(* Logix 5000 project; controller cal1615 1756-L62 rev 20.19; software revision 20.05; part 34 of 82 *)
(* tags used below, declared in another part *)
   aaa_prs : REAL;
   FAULT : BOOL;   // Fault AFI
   HMI : BOOL;   // AFI HMI
   p01r09_pb_global_reset : BOOL;   // System Modes PB: Global Fault Reset
   p19_ai_prs : REAL;   // Advanced Cooling Analog Input Pressure [PSI]
   p19_ai_tc01 : REAL;   // Advanced Cooling Analog Input Control Temperature 1
   p19_ao_cv : REAL;   // Advanced Cooling Analog Output Control Valve
   p19_di_tc01_bo : BOOL;   // Advanced Cooling Digital Input Control Thermocouple 1 Failure
   p19_di_tc02_bo : BOOL;   // Advanced Cooling Digital Input Control Thermocouple 2 Failure
   p19_dint_to_hmi : DINT[16];
   p19_do_pump : BOOL;   // Advanced Cooling Digital Output Enable Pump
   p19_flow_input_max : REAL;
   p19_flow_input_min : REAL;
   p19_flow_output_max : REAL;
   p19_flow_output_min : REAL;
   p19_param_pid2_ff : REAL;
   p19_param_pid2_kd : REAL;
   p19_param_pid2_ki : REAL;
   p19_param_pid2_kp : REAL;
   p19_param_tc01_dev : REAL;
   p19_param_tc01z : REAL;   // Advanced Cooling Parameter Control Temperature 1 Zero Offset
   p19_param_tc02z : REAL;   // Advanced Cooling Parameter Control Temperature 2 Zero Offset
   p19_param_zone_pressure : REAL;   // Advanced Cooling Parameter Minimum Pressusre
   p19_prs_input_max1 : REAL;
   p19_prs_input_min1 : REAL;
   p19_prs_output_max1 : REAL;
   p19_prs_output_min1 : REAL;
   p19_real_to_hmi : REAL[80];   // Advanced Cooling Real to HMI
   p19r01 : routine;   // Advanced Cooling Main
   p19r03_flow_scp : SYS_SCP;   // Advanced Cooling Output Roll Cooling Flow Control
   p19r03_prs_scp : SYS_SCP;   // Advanced Cooling Output Cooling Pressure Control Valve Output
   p19r04 : routine;   // Advanced Cooling Output
   p19r04_timer_fault : TIMER[4];   // Advanced Cooling Output Fault Delay
   p19r04_timer_warning : TIMER[4];   // Advanced Cooling Output Warning Delay
   p19r05 : routine;   // Advanced Cooling Dint to HMI
   p19r05_timer_fault : TIMER[4];   // Advanced Cooing Dint to HMI
   p19r05_timer_warning : TIMER[4];   // Advanced Cooling Dint to HMI Warning Delay
   p19r06 : routine;   // Advanced Cooling Real to HMI
   p19r06_timer_fault : TIMER[4];   // Advanced Cooling Real to HMI Fault Delay
   p19r06_timer_warning : TIMER[4];   // Advanced Cooling Real to HMI Warning Delay
   p19r30_cv_man_sp : REAL;   // Advanced Cooling Manual Control Valve Setpoint
   p19r30_pid_temp : PID;   // Advanced Cooling Temperature Control PID
   p19r30_pid_temp_pv : DINT;   // Advanced Cooling Temperature Control PID Process Variable
   p19r30_request_cool : BOOL;   // Advanced Cooling Temperature Control Request Cool
   p19r30_request_manual : BOOL;   // Advanced Cooling Temperature Control Request Manual Control
   p19r31_request_auto_run : BOOL;   // Advanced Cooling Pump Request Auto Run
(* P19_Advanced_Cooling, continued *)

ROUTINE R04_Output   (* ladder *)
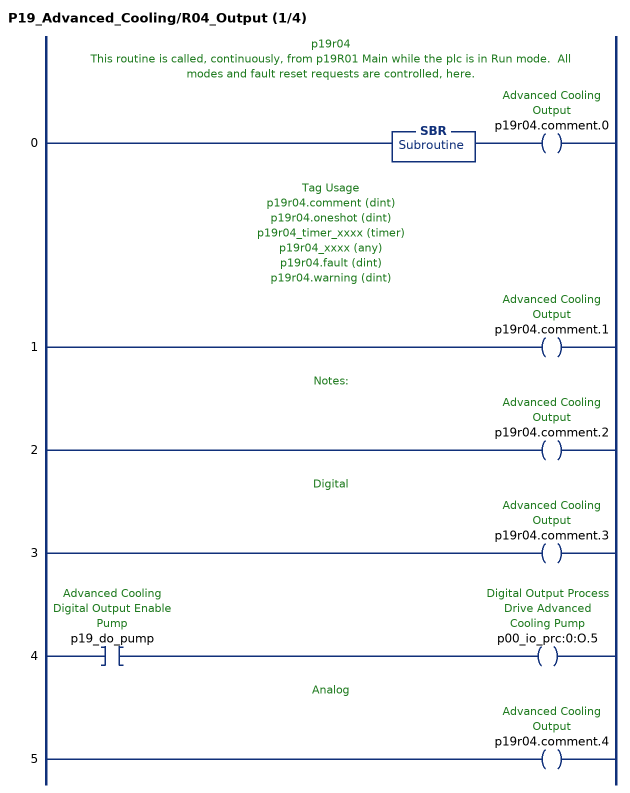
   // p19r04
   // This routine is called, continuously, from p19R01 Main while the plc is in Run mode.  All modes and fault reset requests are controlled, here.
   0: SBR()OTE(p19r04.comment.0);
   // Tag Usage
   // p19r04.comment (dint)
   // p19r04.oneshot (dint)
   // p19r04_timer_xxxx (timer)
   // p19r04_xxxx (any)
   // p19r04.fault (dint)
   // p19r04.warning (dint)
   1: OTE(p19r04.comment.1);
   // Notes:
   2: OTE(p19r04.comment.2);
   // Digital
   3: OTE(p19r04.comment.3);
   4: XIC(p19_do_pump)OTE(p00_io_prc:0:O.5);
   // Analog
   5: OTE(p19r04.comment.4);
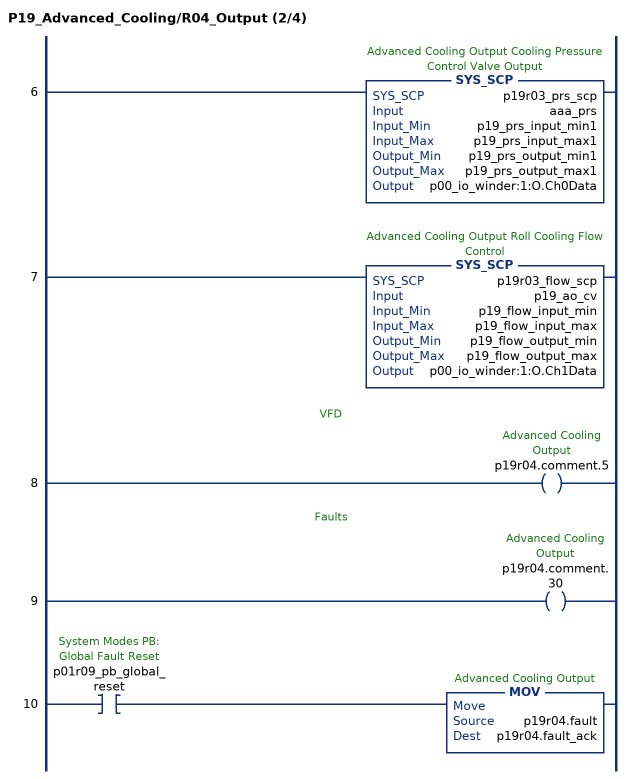
   6: SYS_SCP(p19r03_prs_scp,aaa_prs,p19_prs_input_min1,p19_prs_input_max1,p19_prs_output_min1,p19_prs_output_max1,p00_io_winder:1:O.Ch0Data);
   7: SYS_SCP(p19r03_flow_scp,p19_ao_cv,p19_flow_input_min,p19_flow_input_max,p19_flow_output_min,p19_flow_output_max,p00_io_winder:1:O.Ch1Data);
   // VFD
   8: OTE(p19r04.comment.5);
   // Faults
   9: OTE(p19r04.comment.30);
   10: XIC(p01r09_pb_global_reset)MOV(p19r04.fault,p19r04.fault_ack);
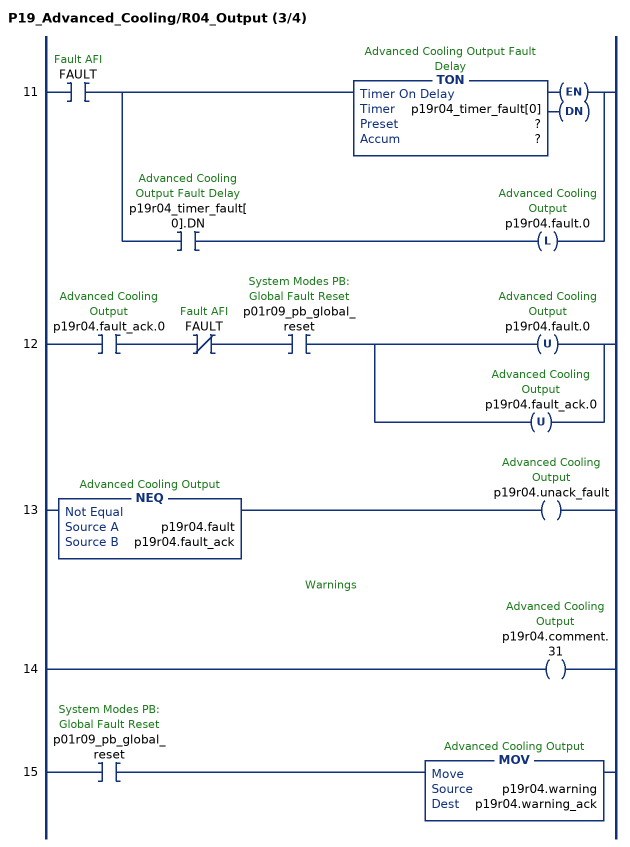
   11: XIC(FAULT)[TON(p19r04_timer_fault[0],?,?) ,XIC(p19r04_timer_fault[0].DN) OTL(p19r04.fault.0) ];
   12: XIC(p19r04.fault_ack.0)XIO(FAULT)XIC(p01r09_pb_global_reset)[OTU(p19r04.fault.0) ,OTU(p19r04.fault_ack.0) ];
   13: NEQ(p19r04.fault,p19r04.fault_ack)OTE(p19r04.unack_fault);
   // Warnings
   14: OTE(p19r04.comment.31);
   15: XIC(p01r09_pb_global_reset)MOV(p19r04.warning,p19r04.warning_ack);
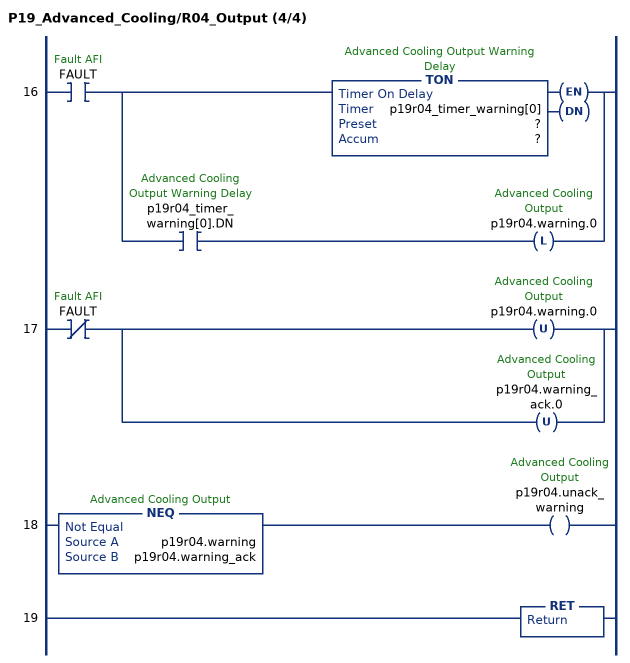
   16: XIC(FAULT)[TON(p19r04_timer_warning[0],?,?) ,XIC(p19r04_timer_warning[0].DN) OTL(p19r04.warning.0) ];
   17: XIO(FAULT)[OTU(p19r04.warning.0) ,OTU(p19r04.warning_ack.0) ];
   18: NEQ(p19r04.warning,p19r04.warning_ack)OTE(p19r04.unack_warning);
   19: RET();
END_ROUTINE

ROUTINE R05_Dint_to_HMI   (* ladder *)
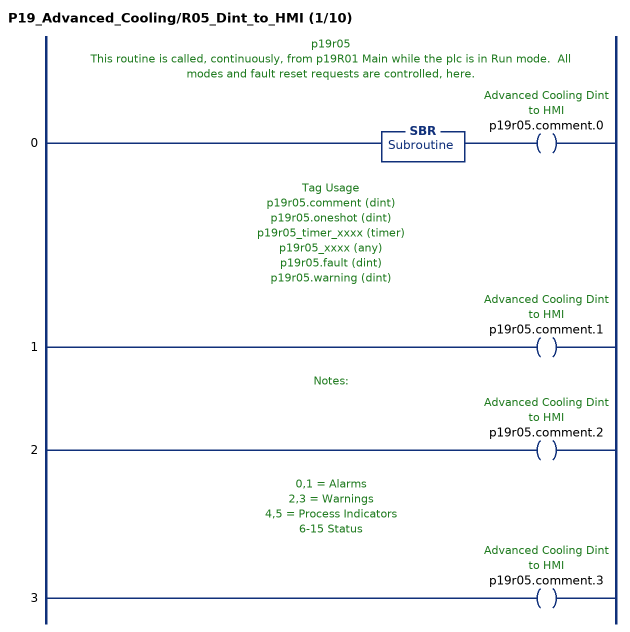
   // p19r05
   // This routine is called, continuously, from p19R01 Main while the plc is in Run mode.  All modes and fault reset requests are controlled, here.
   0: SBR()OTE(p19r05.comment.0);
   // Tag Usage
   // p19r05.comment (dint)
   // p19r05.oneshot (dint)
   // p19r05_timer_xxxx (timer)
   // p19r05_xxxx (any)
   // p19r05.fault (dint)
   // p19r05.warning (dint)
   1: OTE(p19r05.comment.1);
   // Notes:
   2: OTE(p19r05.comment.2);
   // 0,1 = Alarms
   // 2,3 = Warnings
   // 4,5 = Process Indicators
   // 6-15 Status
   3: OTE(p19r05.comment.3);
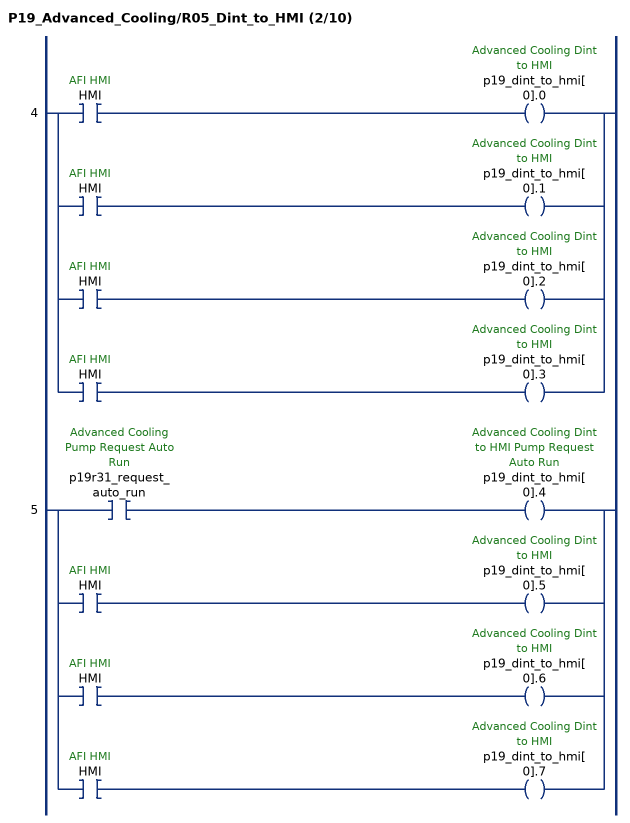
   4: [XIC(HMI) OTE(p19_dint_to_hmi[0].0) ,XIC(HMI) OTE(p19_dint_to_hmi[0].1) ,XIC(HMI) OTE(p19_dint_to_hmi[0].2) ,XIC(HMI) OTE(p19_dint_to_hmi[0].3) ];
   5: [XIC(p19r31_request_auto_run) OTE(p19_dint_to_hmi[0].4) ,XIC(HMI) OTE(p19_dint_to_hmi[0].5) ,XIC(HMI) OTE(p19_dint_to_hmi[0].6) ,XIC(HMI) OTE(p19_dint_to_hmi[0].7) ];
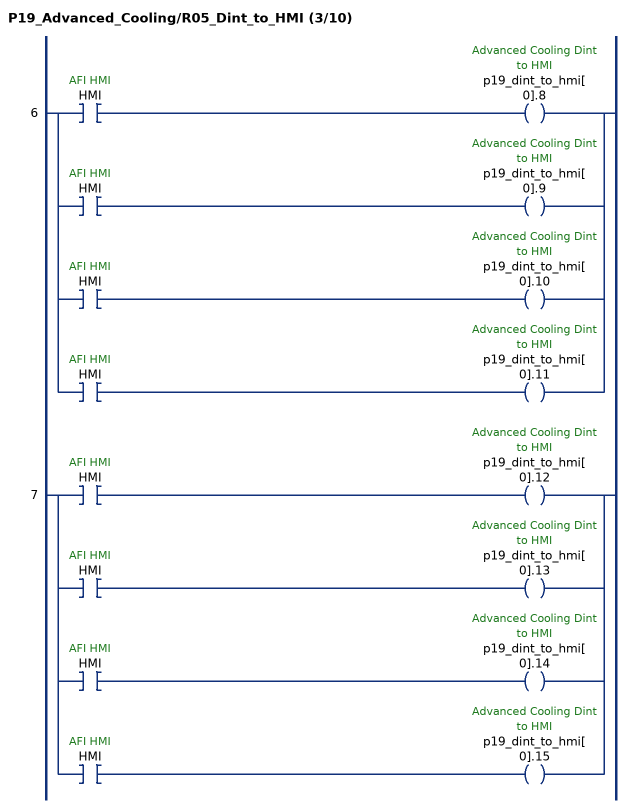
   6: [XIC(HMI) OTE(p19_dint_to_hmi[0].8) ,XIC(HMI) OTE(p19_dint_to_hmi[0].9) ,XIC(HMI) OTE(p19_dint_to_hmi[0].10) ,XIC(HMI) OTE(p19_dint_to_hmi[0].11) ];
   7: [XIC(HMI) OTE(p19_dint_to_hmi[0].12) ,XIC(HMI) OTE(p19_dint_to_hmi[0].13) ,XIC(HMI) OTE(p19_dint_to_hmi[0].14) ,XIC(HMI) OTE(p19_dint_to_hmi[0].15) ];
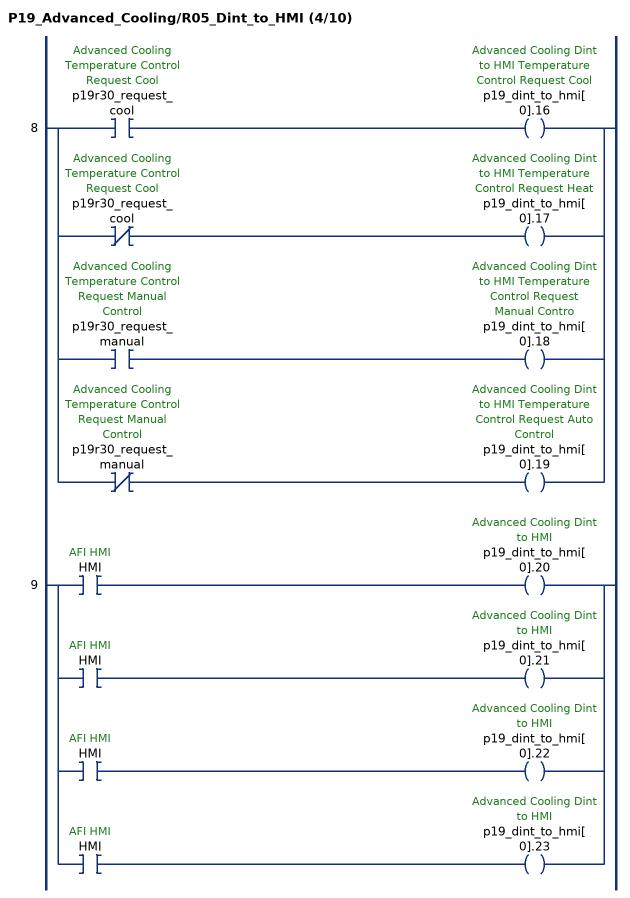
   8: [XIC(p19r30_request_cool) OTE(p19_dint_to_hmi[0].16) ,XIO(p19r30_request_cool) OTE(p19_dint_to_hmi[0].17) ,XIC(p19r30_request_manual) OTE(p19_dint_to_hmi[0].18) ,XIO(p19r30_request_manual) OTE(p19_dint_to_hmi[0].19) ];
   9: [XIC(HMI) OTE(p19_dint_to_hmi[0].20) ,XIC(HMI) OTE(p19_dint_to_hmi[0].21) ,XIC(HMI) OTE(p19_dint_to_hmi[0].22) ,XIC(HMI) OTE(p19_dint_to_hmi[0].23) ];
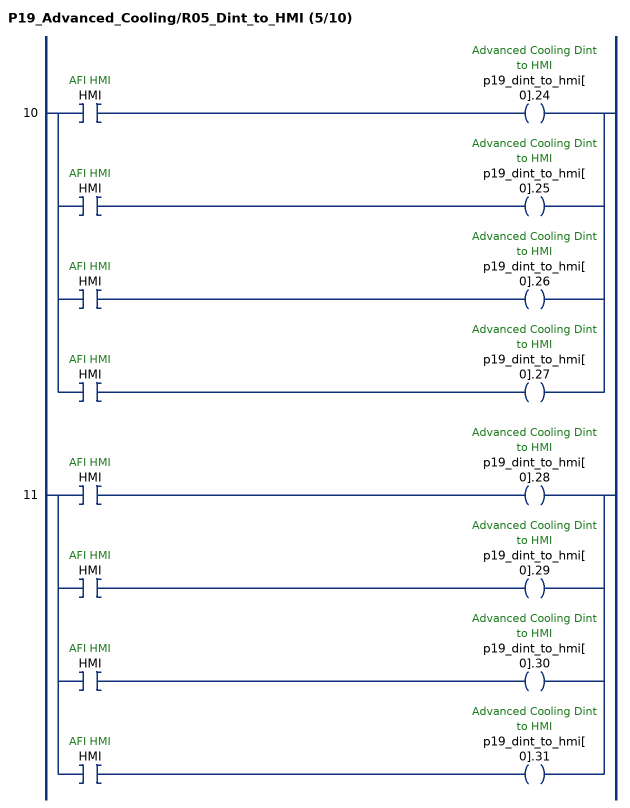
   10: [XIC(HMI) OTE(p19_dint_to_hmi[0].24) ,XIC(HMI) OTE(p19_dint_to_hmi[0].25) ,XIC(HMI) OTE(p19_dint_to_hmi[0].26) ,XIC(HMI) OTE(p19_dint_to_hmi[0].27) ];
   11: [XIC(HMI) OTE(p19_dint_to_hmi[0].28) ,XIC(HMI) OTE(p19_dint_to_hmi[0].29) ,XIC(HMI) OTE(p19_dint_to_hmi[0].30) ,XIC(HMI) OTE(p19_dint_to_hmi[0].31) ];
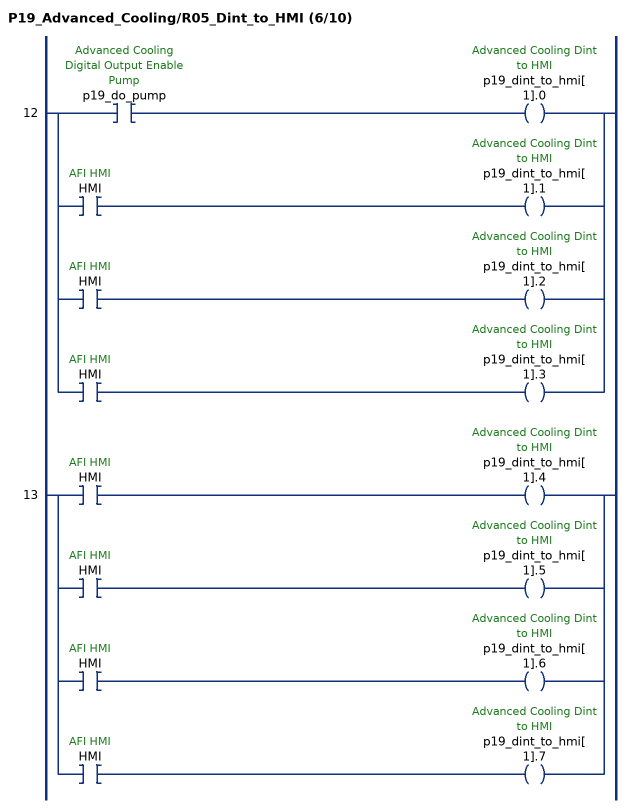
   12: [XIC(p19_do_pump) OTE(p19_dint_to_hmi[1].0) ,XIC(HMI) OTE(p19_dint_to_hmi[1].1) ,XIC(HMI) OTE(p19_dint_to_hmi[1].2) ,XIC(HMI) OTE(p19_dint_to_hmi[1].3) ];
   13: [XIC(HMI) OTE(p19_dint_to_hmi[1].4) ,XIC(HMI) OTE(p19_dint_to_hmi[1].5) ,XIC(HMI) OTE(p19_dint_to_hmi[1].6) ,XIC(HMI) OTE(p19_dint_to_hmi[1].7) ];
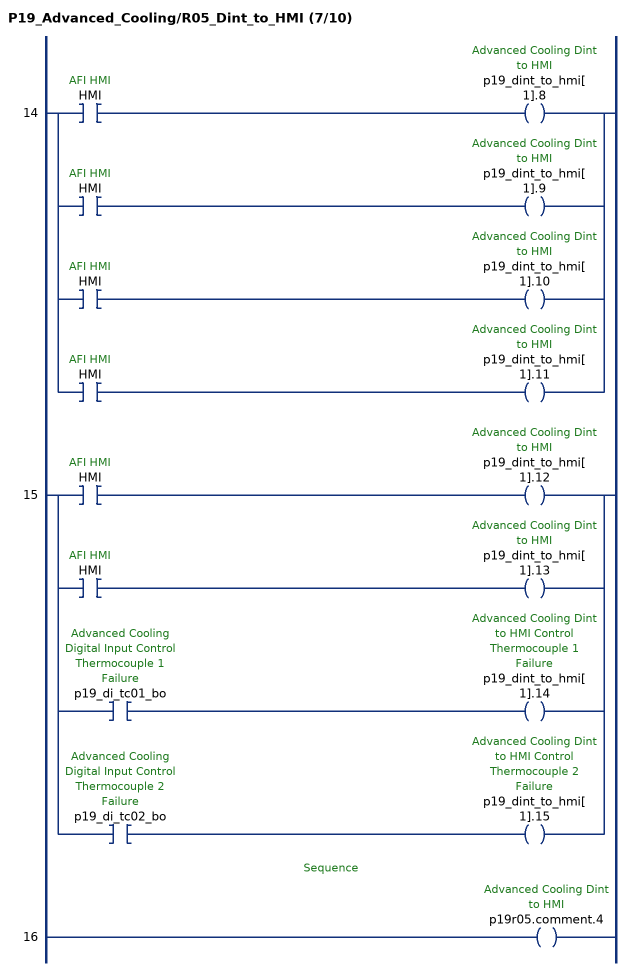
   14: [XIC(HMI) OTE(p19_dint_to_hmi[1].8) ,XIC(HMI) OTE(p19_dint_to_hmi[1].9) ,XIC(HMI) OTE(p19_dint_to_hmi[1].10) ,XIC(HMI) OTE(p19_dint_to_hmi[1].11) ];
   15: [XIC(HMI) OTE(p19_dint_to_hmi[1].12) ,XIC(HMI) OTE(p19_dint_to_hmi[1].13) ,XIC(p19_di_tc01_bo) OTE(p19_dint_to_hmi[1].14) ,XIC(p19_di_tc02_bo) OTE(p19_dint_to_hmi[1].15) ];
   // Sequence
   16: OTE(p19r05.comment.4);
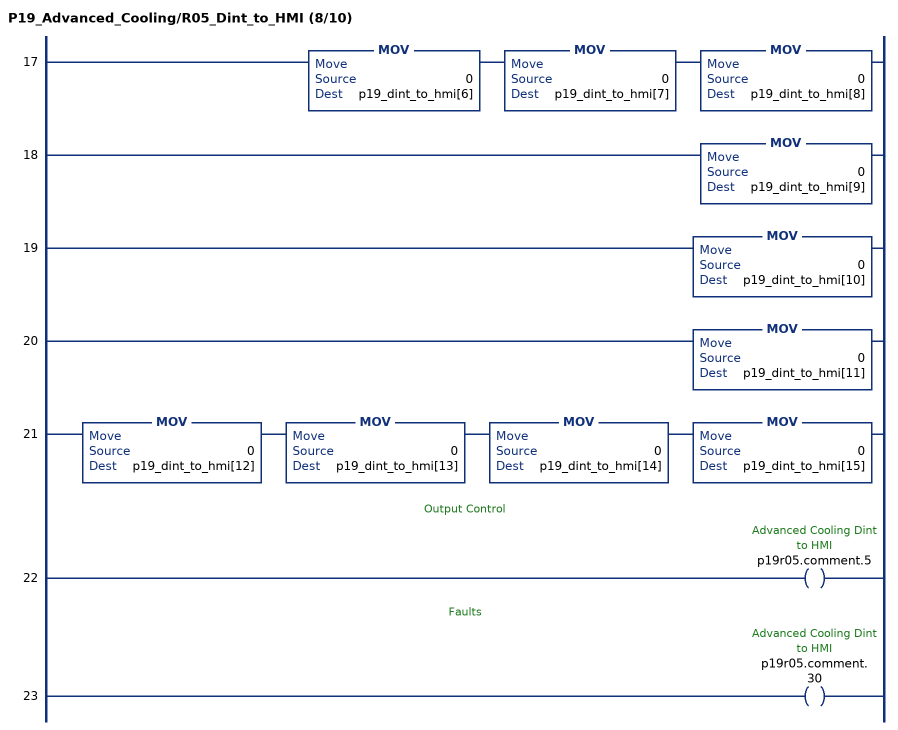
   17: MOV(0,p19_dint_to_hmi[6])MOV(0,p19_dint_to_hmi[7])MOV(0,p19_dint_to_hmi[8]);
   18: MOV(0,p19_dint_to_hmi[9]);
   19: MOV(0,p19_dint_to_hmi[10]);
   20: MOV(0,p19_dint_to_hmi[11]);
   21: MOV(0,p19_dint_to_hmi[12])MOV(0,p19_dint_to_hmi[13])MOV(0,p19_dint_to_hmi[14])MOV(0,p19_dint_to_hmi[15]);
   // Output Control
   22: OTE(p19r05.comment.5);
   // Faults
   23: OTE(p19r05.comment.30);
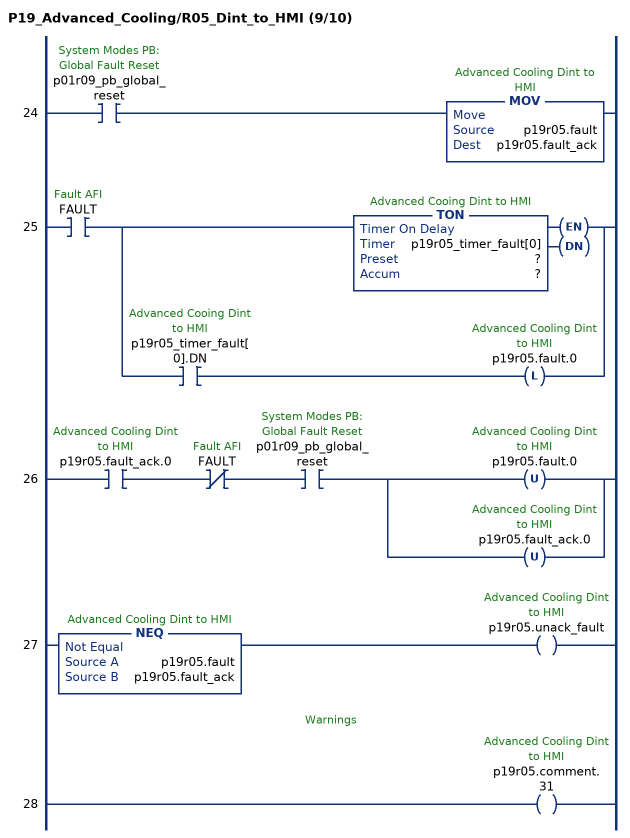
   24: XIC(p01r09_pb_global_reset)MOV(p19r05.fault,p19r05.fault_ack);
   25: XIC(FAULT)[TON(p19r05_timer_fault[0],?,?) ,XIC(p19r05_timer_fault[0].DN) OTL(p19r05.fault.0) ];
   26: XIC(p19r05.fault_ack.0)XIO(FAULT)XIC(p01r09_pb_global_reset)[OTU(p19r05.fault.0) ,OTU(p19r05.fault_ack.0) ];
   27: NEQ(p19r05.fault,p19r05.fault_ack)OTE(p19r05.unack_fault);
   // Warnings
   28: OTE(p19r05.comment.31);
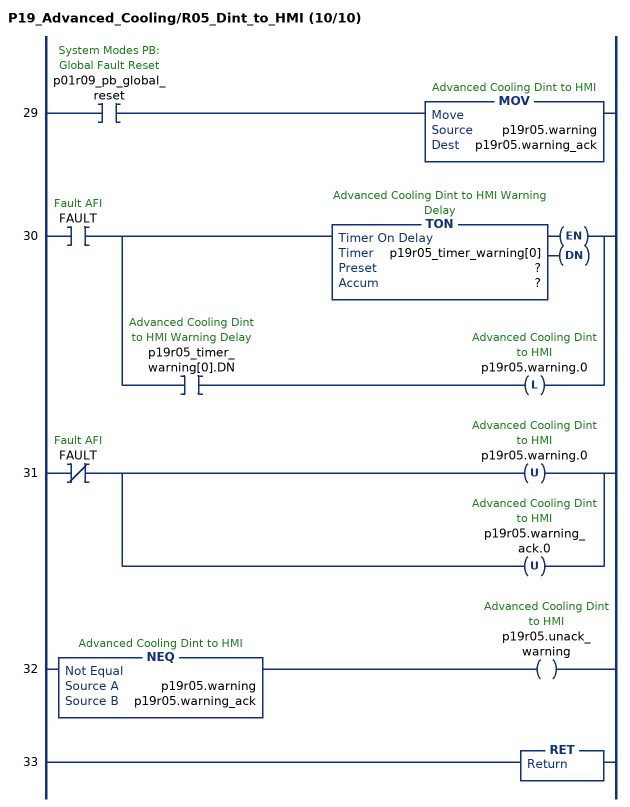
   29: XIC(p01r09_pb_global_reset)MOV(p19r05.warning,p19r05.warning_ack);
   30: XIC(FAULT)[TON(p19r05_timer_warning[0],?,?) ,XIC(p19r05_timer_warning[0].DN) OTL(p19r05.warning.0) ];
   31: XIO(FAULT)[OTU(p19r05.warning.0) ,OTU(p19r05.warning_ack.0) ];
   32: NEQ(p19r05.warning,p19r05.warning_ack)OTE(p19r05.unack_warning);
   33: RET();
END_ROUTINE

ROUTINE R06_Real_to_HMI   (* ladder *)
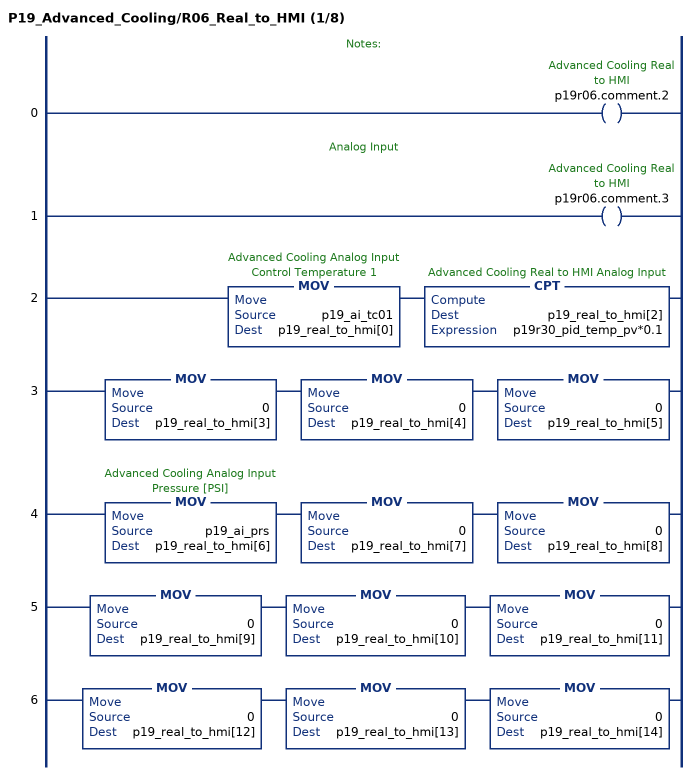
   // Notes:
   0: OTE(p19r06.comment.2);
   // Analog Input
   1: OTE(p19r06.comment.3);
   2: MOV(p19_ai_tc01,p19_real_to_hmi[0])CPT(p19_real_to_hmi[2],p19r30_pid_temp_pv*0.1);
   3: MOV(0,p19_real_to_hmi[3])MOV(0,p19_real_to_hmi[4])MOV(0,p19_real_to_hmi[5]);
   4: MOV(p19_ai_prs,p19_real_to_hmi[6])MOV(0,p19_real_to_hmi[7])MOV(0,p19_real_to_hmi[8]);
   5: MOV(0,p19_real_to_hmi[9])MOV(0,p19_real_to_hmi[10])MOV(0,p19_real_to_hmi[11]);
   6: MOV(0,p19_real_to_hmi[12])MOV(0,p19_real_to_hmi[13])MOV(0,p19_real_to_hmi[14]);
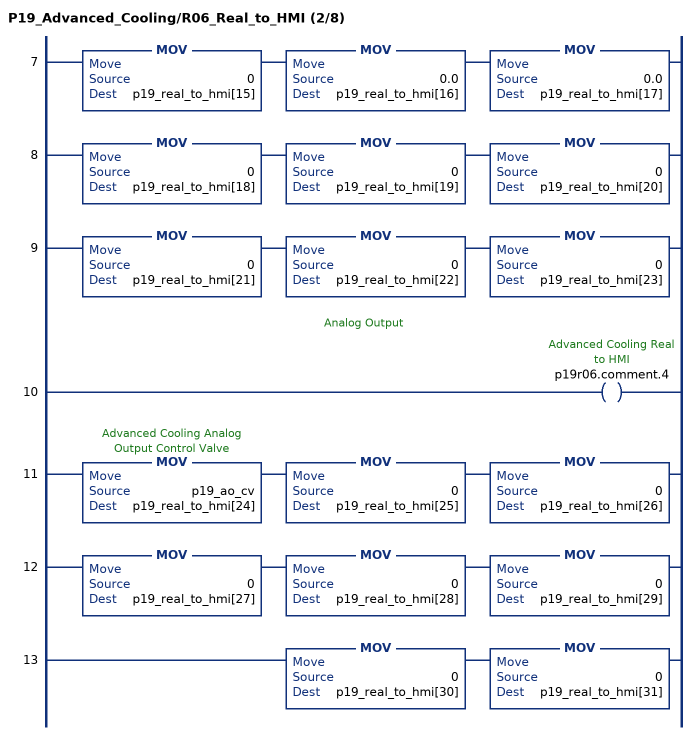
   7: MOV(0,p19_real_to_hmi[15])MOV(0.0,p19_real_to_hmi[16])MOV(0.0,p19_real_to_hmi[17]);
   8: MOV(0,p19_real_to_hmi[18])MOV(0,p19_real_to_hmi[19])MOV(0,p19_real_to_hmi[20]);
   9: MOV(0,p19_real_to_hmi[21])MOV(0,p19_real_to_hmi[22])MOV(0,p19_real_to_hmi[23]);
   // Analog Output
   10: OTE(p19r06.comment.4);
   11: MOV(p19_ao_cv,p19_real_to_hmi[24])MOV(0,p19_real_to_hmi[25])MOV(0,p19_real_to_hmi[26]);
   12: MOV(0,p19_real_to_hmi[27])MOV(0,p19_real_to_hmi[28])MOV(0,p19_real_to_hmi[29]);
   13: MOV(0,p19_real_to_hmi[30])MOV(0,p19_real_to_hmi[31]);
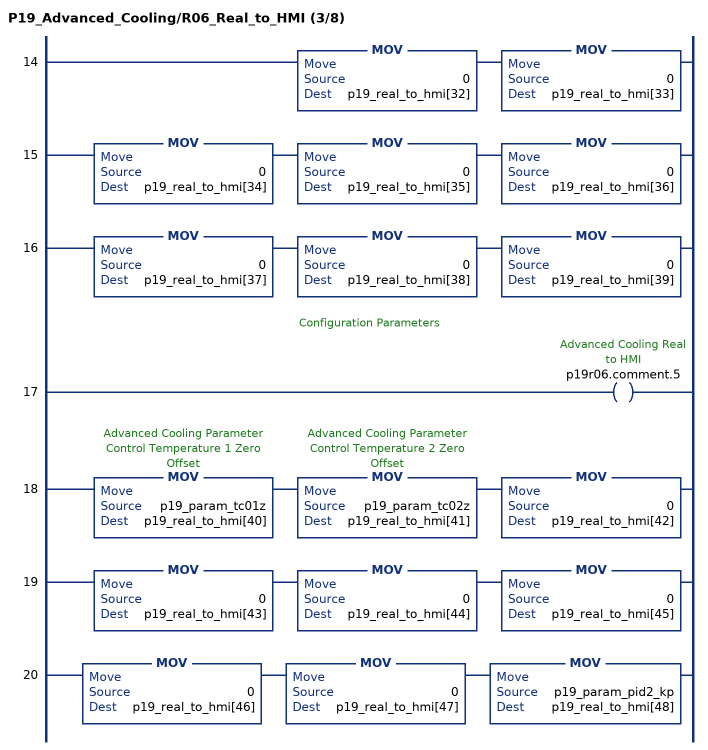
   14: MOV(0,p19_real_to_hmi[32])MOV(0,p19_real_to_hmi[33]);
   15: MOV(0,p19_real_to_hmi[34])MOV(0,p19_real_to_hmi[35])MOV(0,p19_real_to_hmi[36]);
   16: MOV(0,p19_real_to_hmi[37])MOV(0,p19_real_to_hmi[38])MOV(0,p19_real_to_hmi[39]);
   // Configuration Parameters
   17: OTE(p19r06.comment.5);
   18: MOV(p19_param_tc01z,p19_real_to_hmi[40])MOV(p19_param_tc02z,p19_real_to_hmi[41])MOV(0,p19_real_to_hmi[42]);
   19: MOV(0,p19_real_to_hmi[43])MOV(0,p19_real_to_hmi[44])MOV(0,p19_real_to_hmi[45]);
   20: MOV(0,p19_real_to_hmi[46])MOV(0,p19_real_to_hmi[47])MOV(p19_param_pid2_kp,p19_real_to_hmi[48]);
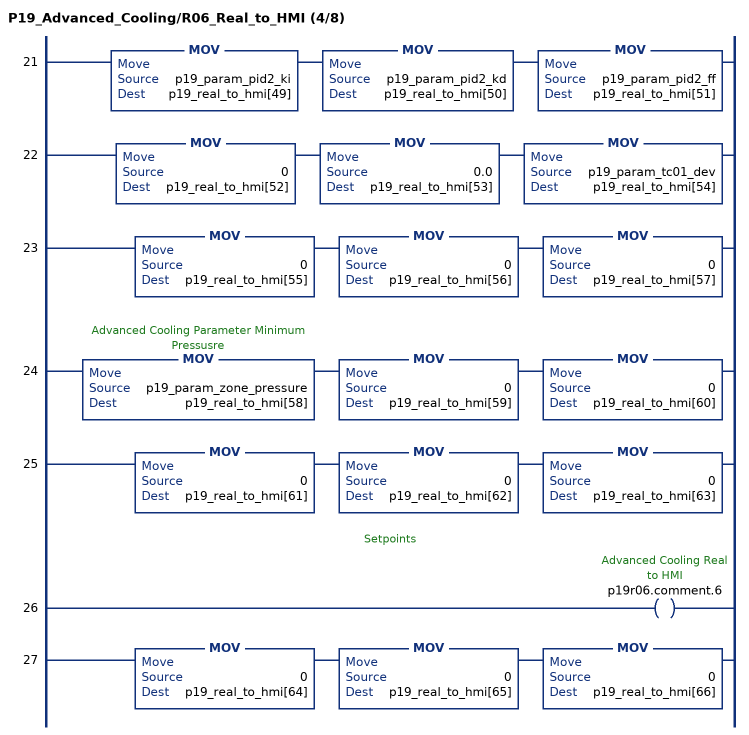
   21: MOV(p19_param_pid2_ki,p19_real_to_hmi[49])MOV(p19_param_pid2_kd,p19_real_to_hmi[50])MOV(p19_param_pid2_ff,p19_real_to_hmi[51]);
   22: MOV(0,p19_real_to_hmi[52])MOV(0.0,p19_real_to_hmi[53])MOV(p19_param_tc01_dev,p19_real_to_hmi[54]);
   23: MOV(0,p19_real_to_hmi[55])MOV(0,p19_real_to_hmi[56])MOV(0,p19_real_to_hmi[57]);
   24: MOV(p19_param_zone_pressure,p19_real_to_hmi[58])MOV(0,p19_real_to_hmi[59])MOV(0,p19_real_to_hmi[60]);
   25: MOV(0,p19_real_to_hmi[61])MOV(0,p19_real_to_hmi[62])MOV(0,p19_real_to_hmi[63]);
   // Setpoints
   26: OTE(p19r06.comment.6);
   27: MOV(0,p19_real_to_hmi[64])MOV(0,p19_real_to_hmi[65])MOV(0,p19_real_to_hmi[66]);
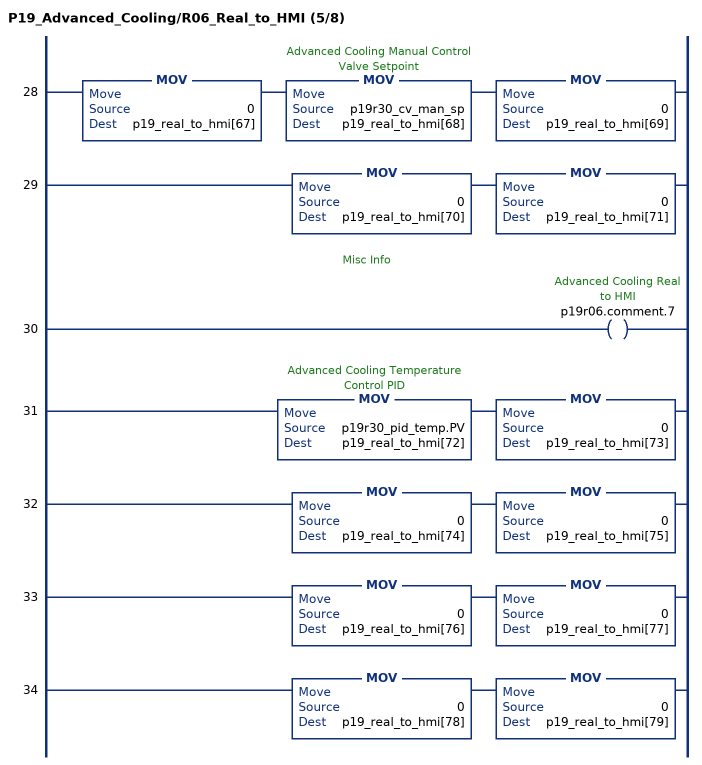
   28: MOV(0,p19_real_to_hmi[67])MOV(p19r30_cv_man_sp,p19_real_to_hmi[68])MOV(0,p19_real_to_hmi[69]);
   29: MOV(0,p19_real_to_hmi[70])MOV(0,p19_real_to_hmi[71]);
   // Misc Info
   30: OTE(p19r06.comment.7);
   31: MOV(p19r30_pid_temp.PV,p19_real_to_hmi[72])MOV(0,p19_real_to_hmi[73]);
   32: MOV(0,p19_real_to_hmi[74])MOV(0,p19_real_to_hmi[75]);
   33: MOV(0,p19_real_to_hmi[76])MOV(0,p19_real_to_hmi[77]);
   34: MOV(0,p19_real_to_hmi[78])MOV(0,p19_real_to_hmi[79]);
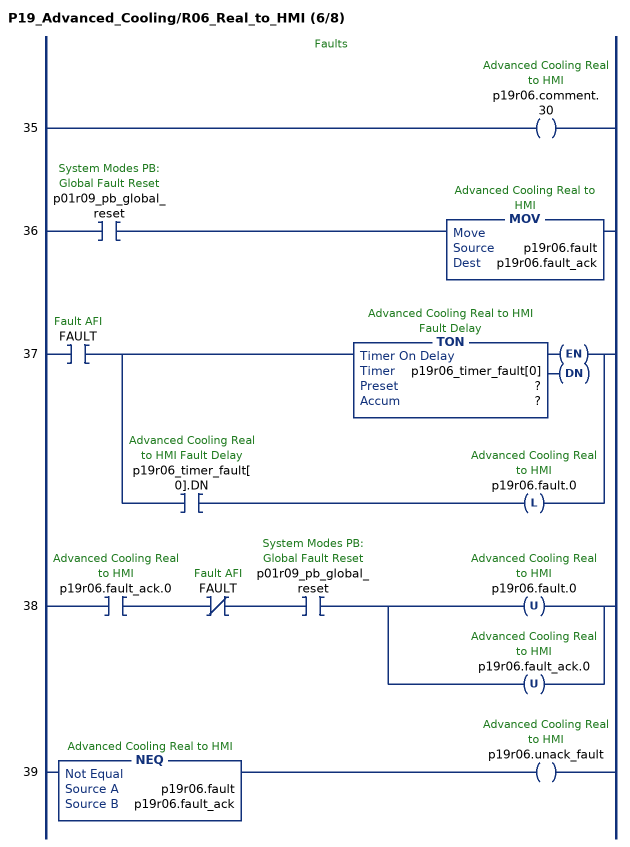
   // Faults
   35: OTE(p19r06.comment.30);
   36: XIC(p01r09_pb_global_reset)MOV(p19r06.fault,p19r06.fault_ack);
   37: XIC(FAULT)[TON(p19r06_timer_fault[0],?,?) ,XIC(p19r06_timer_fault[0].DN) OTL(p19r06.fault.0) ];
   38: XIC(p19r06.fault_ack.0)XIO(FAULT)XIC(p01r09_pb_global_reset)[OTU(p19r06.fault.0) ,OTU(p19r06.fault_ack.0) ];
   39: NEQ(p19r06.fault,p19r06.fault_ack)OTE(p19r06.unack_fault);
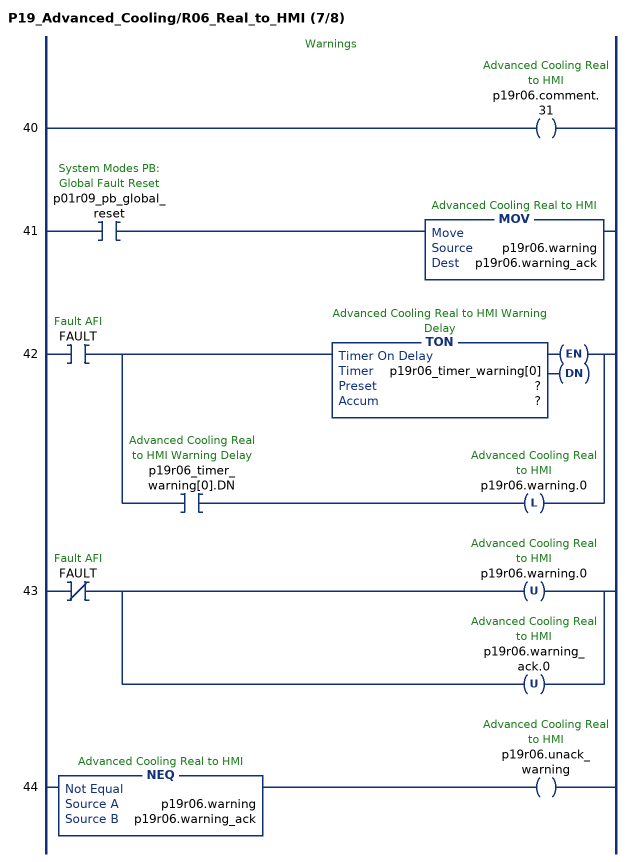
   // Warnings
   40: OTE(p19r06.comment.31);
   41: XIC(p01r09_pb_global_reset)MOV(p19r06.warning,p19r06.warning_ack);
   42: XIC(FAULT)[TON(p19r06_timer_warning[0],?,?) ,XIC(p19r06_timer_warning[0].DN) OTL(p19r06.warning.0) ];
   43: XIO(FAULT)[OTU(p19r06.warning.0) ,OTU(p19r06.warning_ack.0) ];
   44: NEQ(p19r06.warning,p19r06.warning_ack)OTE(p19r06.unack_warning);
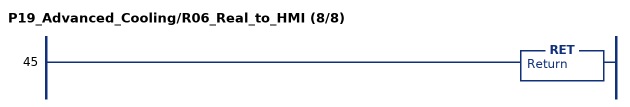
   45: RET();
END_ROUTINE
